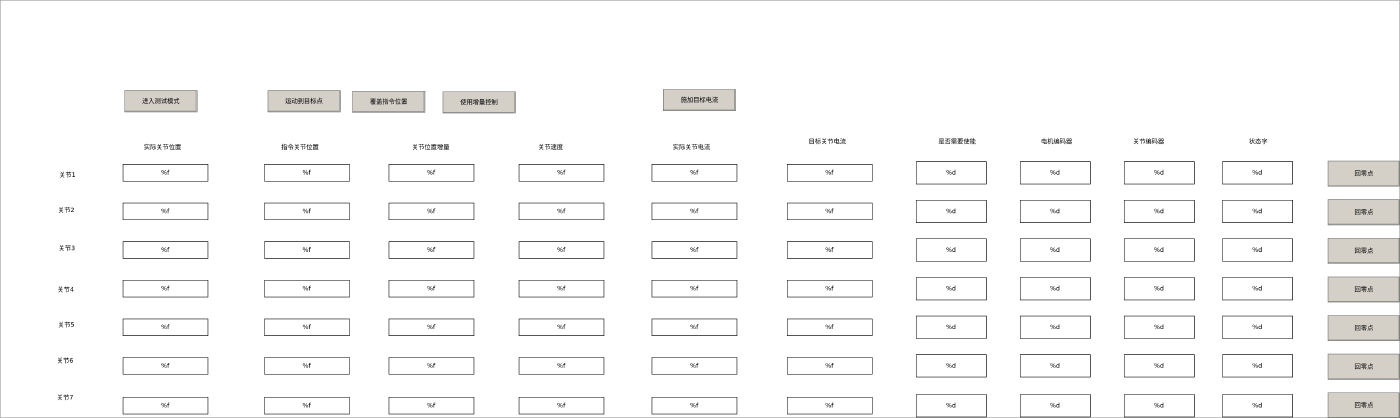
VISUALIZATION motion_a1  // 2464x736
    Label (211,244 150x30), "实际关节位置"
    Rectangle (216,289 150x30), "%f", text variable: g_motionTest.m_armActJntPos[1][1]
    Label (453,244 150x30), "指令关节位置"
    Button (219,159 128x38), "进入测试模式", colour toggle: g_motionTest.m_enterPrecisionTestMode[1]
        toggle g_motionTest.m_enterPrecisionTestMode[1]
    Button (471,159 128x38), "运动到目标点", colour toggle: g_motionTest.m_uiArmMode[1,1]
        tap g_motionTest.m_uiArmMode[1,1]
    Label (683,244 150x30), "关节位置增量"
    Rectangle (684,289 150x30), "%f", text variable: g_motionTest.m_targetJntPosInc[1][1]
        OnMouseClick: write the text variable via Default
    Label (1142,244 150x30), "实际关节电流"
    Rectangle (1147,289 150x30), "%f", text variable: g_motionTest.m_curJntCurrent[1][1]
    Label (1381,234 150x30), "目标关节电流"
    Rectangle (1385,289 150x30), "%f", text variable: g_motionTest.m_targetJntCurrent[1][1]
        OnMouseClick: write the text variable via Default
    Button (1167,157 128x38), "施加目标电流", colour toggle: g_motionTest.m_uiArmMode[1,8]
        toggle g_motionTest.m_uiArmMode[1,8]
    Rectangle (216,357 150x30), "%f", text variable: g_motionTest.m_armActJntPos[1][2]
    Rectangle (216,425 150x30), "%f", text variable: g_motionTest.m_armActJntPos[1][3]
    Rectangle (216,493 150x30), "%f", text variable: g_motionTest.m_armActJntPos[1][4]
    Rectangle (216,561 150x30), "%f", text variable: g_motionTest.m_armActJntPos[1][5]
    Rectangle (216,629 150x30), "%f", text variable: g_motionTest.m_armActJntPos[1][6]
    Rectangle (216,699 150x30), "%f", text variable: g_motionTest.m_armActJntPos[1][7]
    Rectangle (465,289 150x30), "%f", text variable: g_motionTest.m_targetJntPos[1][1]
        OnMouseClick: write the text variable via Default
    Rectangle (465,357 150x30), "%f", text variable: g_motionTest.m_targetJntPos[1][2]
        OnMouseClick: write the text variable via Default
    Rectangle (465,425 150x30), "%f", text variable: g_motionTest.m_targetJntPos[1][3]
        OnMouseClick: write the text variable via Default
    Rectangle (465,493 150x30), "%f", text variable: g_motionTest.m_targetJntPos[1][4]
        OnMouseClick: write the text variable via Default
    Rectangle (465,561 150x30), "%f", text variable: g_motionTest.m_targetJntPos[1][5]
        OnMouseClick: write the text variable via Default
    Rectangle (465,629 150x30), "%f", text variable: g_motionTest.m_targetJntPos[1][6]
        OnMouseClick: write the text variable via Default
    Rectangle (465,699 150x30), "%f", text variable: g_motionTest.m_targetJntPos[1][7]
        OnMouseClick: write the text variable via Default
    Button (779,161 128x38), "使用增量控制", colour toggle: g_motionTest.m_jntPosIncMode[1]
        toggle g_motionTest.m_jntPosIncMode[1]
    Rectangle (684,357 150x30), "%f", text variable: g_motionTest.m_targetJntPosInc[1][2]
        OnMouseClick: write the text variable via Default
    Rectangle (684,425 150x30), "%f", text variable: g_motionTest.m_targetJntPosInc[1][3]
        OnMouseClick: write the text variable via Default
    Rectangle (684,493 150x30), "%f", text variable: g_motionTest.m_targetJntPosInc[1][4]
        OnMouseClick: write the text variable via Default
    Rectangle (684,561 150x30), "%f", text variable: g_motionTest.m_targetJntPosInc[1][5]
        OnMouseClick: write the text variable via Default
    Rectangle (684,629 150x30), "%f", text variable: g_motionTest.m_targetJntPosInc[1][6]
        OnMouseClick: write the text variable via Default
    Rectangle (684,699 150x30), "%f", text variable: g_motionTest.m_targetJntPosInc[1][7]
        OnMouseClick: write the text variable via Default
    Rectangle (1385,357 150x30), "%f", text variable: g_motionTest.m_targetJntCurrent[1][2]
        OnMouseClick: write the text variable via Default
    Rectangle (1385,425 150x30), "%f", text variable: g_motionTest.m_targetJntCurrent[1][3]
        OnMouseClick: write the text variable via Default
    Rectangle (1385,493 150x30), "%f", text variable: g_motionTest.m_targetJntCurrent[1][4]
        OnMouseClick: write the text variable via Default
    Rectangle (1385,561 150x30), "%f", text variable: g_motionTest.m_targetJntCurrent[1][5]
        OnMouseClick: write the text variable via Default
    Rectangle (1385,629 150x30), "%f", text variable: g_motionTest.m_targetJntCurrent[1][6]
        OnMouseClick: write the text variable via Default
    Rectangle (1385,699 150x30), "%f", text variable: g_motionTest.m_targetJntCurrent[1][7]
        OnMouseClick: write the text variable via Default
    Rectangle (1147,357 150x30), "%f", text variable: g_motionTest.m_curJntCurrent[1][2]
    Rectangle (1147,425 150x30), "%f", text variable: g_motionTest.m_curJntCurrent[1][3]
    Rectangle (1147,493 150x30), "%f", text variable: g_motionTest.m_curJntCurrent[1][4]
    Rectangle (1147,561 150x30), "%f", text variable: g_motionTest.m_curJntCurrent[1][5]
    Rectangle (1147,629 150x30), "%f", text variable: g_motionTest.m_curJntCurrent[1][6]
    Rectangle (1147,699 150x30), "%f", text variable: g_motionTest.m_curJntCurrent[1][7]
    Label (894,244 150x30), "关节速度"
    Rectangle (913,289 150x30), "%f", text variable: g_motionTest.m_targetJntVel[1][1]
        OnMouseClick: write the text variable via Default
    Rectangle (913,357 150x30), "%f", text variable: g_motionTest.m_targetJntVel[1][2]
        OnMouseClick: write the text variable via Default
    Rectangle (913,425 150x30), "%f", text variable: g_motionTest.m_targetJntVel[1][3]
        OnMouseClick: write the text variable via Default
    Rectangle (913,493 150x30), "%f", text variable: g_motionTest.m_targetJntVel[1][4]
        OnMouseClick: write the text variable via Default
    Rectangle (913,561 150x30), "%f", text variable: g_motionTest.m_targetJntVel[1][5]
        OnMouseClick: write the text variable via Default
    Rectangle (913,629 150x30), "%f", text variable: g_motionTest.m_targetJntVel[1][6]
        OnMouseClick: write the text variable via Default
    Rectangle (913,699 150x30), "%f", text variable: g_motionTest.m_targetJntVel[1][7]
        OnMouseClick: write the text variable via Default
    Label (1612,234 145x30), "是否需要使能"
    Rectangle (1612,284 124x40), "%d", text variable: g_motionTest.m_jntEnable[1][1]
        OnMouseClick: write the text variable via Default
    Rectangle (1612,352 124x40), "%d", text variable: g_motionTest.m_jntEnable[1][2]
        OnMouseClick: write the text variable via Default
    Rectangle (1612,420 124x40), "%d", text variable: g_motionTest.m_jntEnable[1][3]
        OnMouseClick: write the text variable via Default
    Rectangle (1612,488 124x40), "%d", text variable: g_motionTest.m_jntEnable[1][4]
        OnMouseClick: write the text variable via Default
    Rectangle (1612,556 124x40), "%d", text variable: g_motionTest.m_jntEnable[1][5]
        OnMouseClick: write the text variable via Default
    Rectangle (1612,624 124x40), "%d", text variable: g_motionTest.m_jntEnable[1][6]
        OnMouseClick: write the text variable via Default
    Rectangle (1612,694 124x40), "%d", text variable: g_motionTest.m_jntEnable[1][7]
        OnMouseClick: write the text variable via Default
    Label (1787,235 145x28), "电机编码器"
    Label (1949,235 145x28), "关节编码器"
    Label (2142,235 145x28), "状态字"
    Rectangle (1795,284 124x40), "%d", text variable: g_systemInfo.m_armJntInfo[1,1].m_motorInput.m_motorEncoder
    Rectangle (1795,352 124x40), "%d", text variable: g_systemInfo.m_armJntInfo[1,2].m_motorInput.m_motorEncoder
    Rectangle (1795,420 124x40), "%d", text variable: g_systemInfo.m_armJntInfo[1,3].m_motorInput.m_motorEncoder
    Rectangle (1795,488 124x40), "%d", text variable: g_systemInfo.m_armJntInfo[1,4].m_motorInput.m_motorEncoder
    Rectangle (1795,556 124x40), "%d", text variable: g_systemInfo.m_armJntInfo[1,5].m_motorInput.m_motorEncoder
    Rectangle (1795,624 124x40), "%d", text variable: g_systemInfo.m_armJntInfo[1,6].m_motorInput.m_motorEncoder
    Rectangle (1795,694 124x40), "%d", text variable: g_systemInfo.m_armJntInfo[1,7].m_motorInput.m_motorEncoder
    Rectangle (1978,284 124x40), "%d", text variable: g_systemInfo.m_armJntInfo[1,1].m_motorInput.m_linkEncoder
    Rectangle (1978,352 124x40), "%d", text variable: g_systemInfo.m_armJntInfo[1,2].m_motorInput.m_linkEncoder
    Rectangle (1978,420 124x40), "%d", text variable: g_systemInfo.m_armJntInfo[1,3].m_motorInput.m_linkEncoder
    Rectangle (1978,488 124x40), "%d", text variable: g_systemInfo.m_armJntInfo[1,4].m_motorInput.m_linkEncoder
    Rectangle (1978,556 124x40), "%d", text variable: g_systemInfo.m_armJntInfo[1,5].m_motorInput.m_linkEncoder
    Rectangle (1978,624 124x40), "%d", text variable: g_systemInfo.m_armJntInfo[1,6].m_motorInput.m_linkEncoder
    Rectangle (1978,694 124x40), "%d", text variable: g_systemInfo.m_armJntInfo[1,7].m_motorInput.m_linkEncoder
    Rectangle (2151,284 124x40), "%d", text variable: g_systemInfo.m_armJntInfo[1,1].m_motorInput.m_statusWord
    Rectangle (2151,352 124x40), "%d", text variable: g_systemInfo.m_armJntInfo[1,2].m_motorInput.m_statusWord
    Rectangle (2151,420 124x40), "%d", text variable: g_systemInfo.m_armJntInfo[1,3].m_motorInput.m_statusWord
    Rectangle (2151,488 124x40), "%d", text variable: g_systemInfo.m_armJntInfo[1,4].m_motorInput.m_statusWord
    Rectangle (2151,556 124x40), "%d", text variable: g_systemInfo.m_armJntInfo[1,5].m_motorInput.m_statusWord
    Rectangle (2151,624 124x40), "%d", text variable: g_systemInfo.m_armJntInfo[1,6].m_motorInput.m_statusWord
    Rectangle (2151,694 124x40), "%d", text variable: g_systemInfo.m_armJntInfo[1,7].m_motorInput.m_statusWord
    Button (620,160 128x38), "覆盖指令位置", colour toggle: g_motionTest.m_coverCmdPos[1]
        tap g_motionTest.m_coverCmdPos[1]
    Button (2337,283 127x45), "回零点", colour toggle: g_motionTest.m_goHome[1][1]
        tap g_motionTest.m_goHome[1][1]
    Label (67,290 103x36), "关节1"
    Label (65,352 103x36), "关节2"
    Label (66,419 103x36), "关节3"
    Label (64,492 103x36), "关节4"
    Label (65,554 103x36), "关节5"
    Label (63,617 103x36), "关节6"
    Label (63,682 103x36), "关节7"
    Button (2337,351 127x45), "回零点", colour toggle: g_motionTest.m_goHome[1][2]
        tap g_motionTest.m_goHome[1][2]
    Button (2337,419 127x45), "回零点", colour toggle: g_motionTest.m_goHome[1][3]
        tap g_motionTest.m_goHome[1][3]
    Button (2337,487 127x45), "回零点", colour toggle: g_motionTest.m_goHome[1][4]
        tap g_motionTest.m_goHome[1][4]
    Button (2337,555 127x45), "回零点", colour toggle: g_motionTest.m_goHome[1][5]
        tap g_motionTest.m_goHome[1][5]
    Button (2337,623 127x45), "回零点", colour toggle: g_motionTest.m_goHome[1][6]
        tap g_motionTest.m_goHome[1][6]
    Button (2337,691 127x45), "回零点", colour toggle: g_motionTest.m_goHome[1][7]
        tap g_motionTest.m_goHome[1][7]
END_VISUALIZATION

(* stored: Version 1.1.0.1, ProductVersion 3.1.4024.11
   Visu motion_a1: Id {b0f708fb-d056-48d5-9719-2ad7098ee580} *)
